Staubli VAL3: start.pgx

program start()
begin

  //程序入口
  call main()
end
